PROGRAM Main_Send
VAR
END_VAR

//Main_SendData();
Main_SendIMU();
;

END_PROGRAM

(* stored: Version 1.1.0.1, ProductVersion 3.1.4024.6
   POU Main_Send: Id {d7cc139f-c0a0-4426-8778-8d0a6349ccdb}, SpecialFunc None *)
